SUBAPPLICATION Softkey_Aux_Switch_Auto_TO_Remote_WRITE_BG_OPC (* VT-SoftKey lesen ODER AUX-Zuweisung (Joystick) lesen ODER lokaler Web-Override ODER physischer Remote-Taster auf einem dritten Modul ODER Automatik-Kommando + Remote-OPC-UA-Write an Zielmodul + VT-Hintergrundfarbe (SoftKey UND AUX) aus Remote-Subscribe (5-Quellen-Variante von Softkey_Aux_Switch_TO_Remote_WRITE_BG_OPC um einen zusaetzlichen AUTO_IN-Socket, z.B. Fuellband Heben: SoftKey/AUX/Web/physischer Taster S08 UND Befuellautomatik-Hysterese) *)
  (* Standard: 61499-2; Description: Copyright (c) 2026 Meisterschulen am Ostbahnhof This program and the accompanying materials are made available under the terms of the Eclipse Public License 2.0 which is available at https://www.eclipse.org/legal/epl-2.0/ SPDX-License-Identifier: EPL-2.0 *)
  (* Version 1.1, 2026-09-26, Franz Höpfinger, Meisterschulen am Ostbahnhof, Neuer optionaler Plug CMD_OUT, durchgereicht von Command.CMD_OUT (siehe Softkey_Aux_Switch_Auto_TO_Remote_WRITE.SUB v1.1) - rein additiv, bestehende Instanzen unveraendert nutzbar. *)
  (* Version 1.0, 2026-09-13, Franz Höpfinger, Meisterschulen am Ostbahnhof, initial implementation - 5-Quellen-Variante fuer Fuellband Heben (Befuellautomatik, KVE14 Funktionen und Bedingungen Zeile 22). *)
  PACKAGE MyLib::sys;
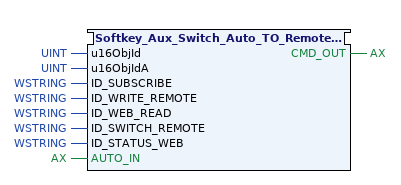
  VAR_INPUT
    u16ObjId : UINT; (* Object ID SoftKey/Hintergrund (VT) *)
    u16ObjIdA : UINT; (* Object ID AuxFunction2/Hintergrund (VT) *)
    ID_SUBSCRIBE : WSTRING; (* Remote-Subscribe-Adresse (Status/Farbe, ACTION=SUBSCRIBE) *)
    ID_WRITE_REMOTE : WSTRING; (* Remote-Write-Adresse zum Zielmodul (Befehl, ACTION=WRITE, CLIENT) *)
    ID_WEB_READ : WSTRING; (* Lokale Subscribe-Adresse fuer einen Web-Client (z.B. vt-ui-mirror) auf demselben Modul, ODER-verknuepft mit SoftKey und AUX *)
    ID_SWITCH_REMOTE : WSTRING; (* Remote-Subscribe-Adresse eines zusaetzlichen physischen Tasters auf einem ANDEREN Modul, ODER-verknuepft mit SoftKey/AUX/Web/Automatik *)
    ID_STATUS_WEB : WSTRING; (* Lokale Publish-Adresse (auf diesem Modul) fuer den vom Zielmodul zurueckgemeldeten Zustand - damit ein Web-Client (z.B. vt-ui-mirror) dieselbe Hintergrundfarbe wie das echte VT zeigen kann *)
  END_VAR
  SOCKETS
    AUTO_IN : adapter::types::unidirectional::AX; (* Autonomes Kommando (z.B. Befuellautomatik-Hysterese), ODER-verknuepft mit SoftKey/Aux/Web/physischem Taster *)
  END_SOCKETS
  PLUGS
    CMD_OUT : adapter::types::unidirectional::AX; (* Optional: lokal gemergter Rohbefehl, durchgereicht von Command.CMD_OUT - unverdrahtet lassen, wenn nicht gebraucht *)
  END_PLUGS
  SUBAPPS
    Command : MyLib::sys::Softkey_Aux_Switch_Auto_TO_Remote_WRITE;
    Status : MyLib::sys::AX_SUBSCRIBE_BG3_WEB_OPC;
  END_SUBAPPS
  DATA_CONNECTIONS
    u16ObjId TO Command.u16ObjId;
    u16ObjIdA TO Command.u16ObjIdA;
    ID_WRITE_REMOTE TO Command.ID_WRITE_REMOTE;
    ID_WEB_READ TO Command.ID_WEB_READ;
    ID_SWITCH_REMOTE TO Command.ID_SWITCH_REMOTE;
    u16ObjId TO Status.u16ObjId;
    u16ObjIdA TO Status.u16ObjIdA;
    ID_SUBSCRIBE TO Status.ID_SUBSCRIBE;
    ID_STATUS_WEB TO Status.ID_STATUS_WEB;
  END_CONNECTIONS
  ADAPTER_CONNECTIONS
    AUTO_IN TO Command.AUTO_IN;
    Command.CMD_OUT TO CMD_OUT;
  END_CONNECTIONS
END_SUBAPPLICATION
